// Mitsubishi GX Works2 project: PLC FX1N Program Awal Bawaan   PLC: FX1N/FX1NC

PROGRAM MAIN
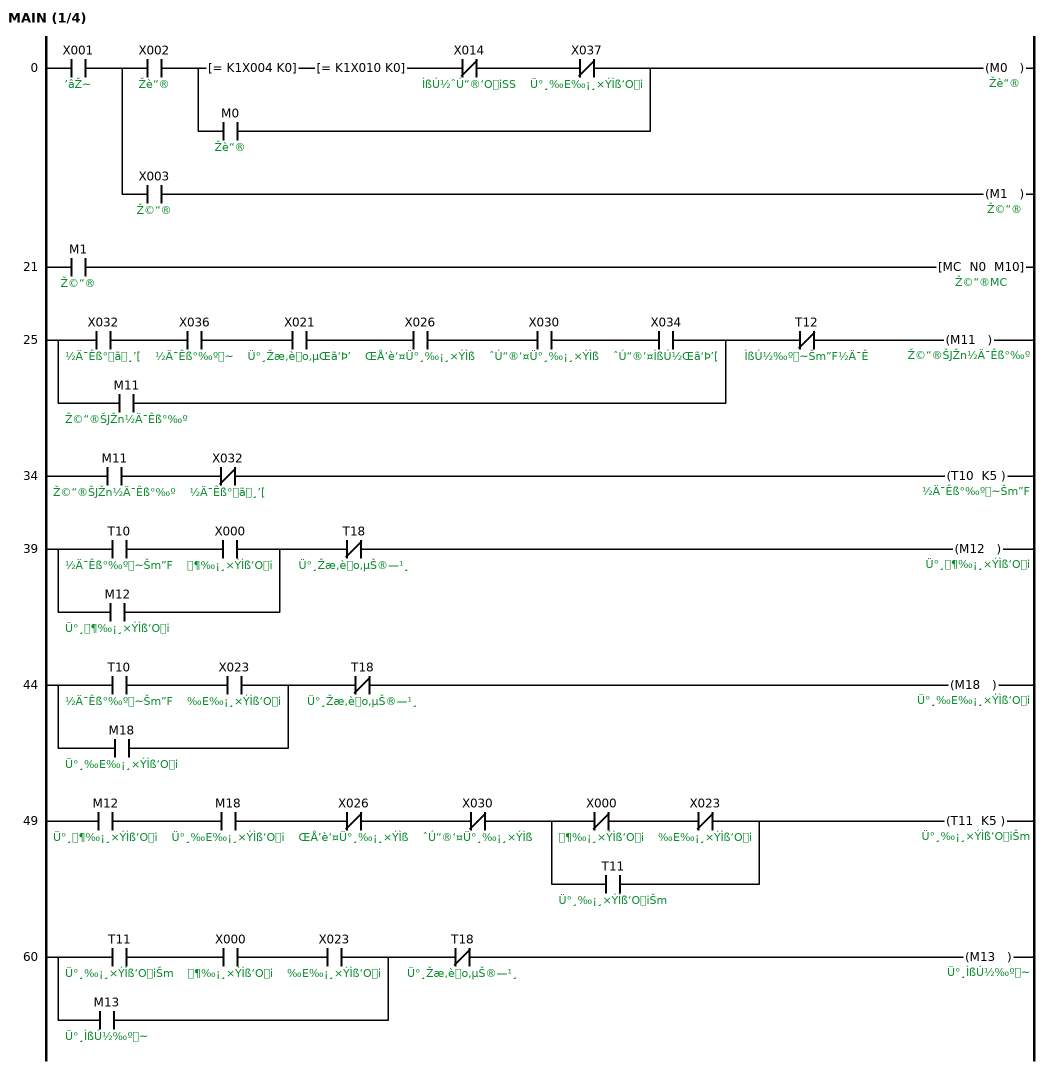
0     LD      X001  ; ’âŽ~
      MPS
      AND     X002  ; Žè“®
      LD=     K1X004 K0  ; Ü°¸Žæ‚èo‚µˆÚ“®‘
      AND=    K1X010 K0  ; ½Ä¯Êß°‰º~SS
      ANI     X014  ; ÌßÚ½ˆÚ“®‘OiSS
      ANI     X037  ; Ü°¸‰E‰¡¸×ÝÌß‘Oi
      OR      M0  ; Žè“®
      ANB
      OUT     M0  ; Žè“®
      MPP
      AND     X003  ; Ž©“®
      OUT     M1  ; Ž©“®
21    LD      M1  ; Ž©“®
      MC      N0 M10  ; Ž©“®MC
25    LD      X032  ; ½Ä¯Êß°ã¸’[
      AND     X036  ; ½Ä¯Êß°‰º~
      AND     X021  ; Ü°¸Žæ‚èo‚µŒã‘Þ’
      AND     X026  ; ŒÅ’è‘¤Ü°¸‰¡¸×ÝÌß
      AND     X030  ; ˆÚ“®‘¤Ü°¸‰¡¸×ÝÌß
      AND     X034  ; ˆÚ“®‘¤ÌßÚ½Œã‘Þ’[
      OR      M11  ; Ž©“®ŠJŽn½Ä¯Êß°‰º
      ANI     T12  ; ÌßÚ½‰º~Šm”F½Ä¯Ê
      OUT     M11  ; Ž©“®ŠJŽn½Ä¯Êß°‰º
34    LD      M11  ; Ž©“®ŠJŽn½Ä¯Êß°‰º
      ANI     X032  ; ½Ä¯Êß°ã¸’[
      OUT     T10 K5  ; ½Ä¯Êß°‰º~Šm”F
39    LD      T10  ; ½Ä¯Êß°‰º~Šm”F
      AND     X000  ; ¶‰¡¸×ÝÌß‘Oi
      OR      M12  ; Ü°¸¶‰¡¸×ÝÌß‘Oi
      ANI     T18  ; Ü°¸Žæ‚èo‚µŠ®—¹¸
      OUT     M12  ; Ü°¸¶‰¡¸×ÝÌß‘Oi
44    LD      T10  ; ½Ä¯Êß°‰º~Šm”F
      AND     X023  ; ‰E‰¡¸×ÝÌß‘Oi
      OR      M18  ; Ü°¸‰E‰¡¸×ÝÌß‘Oi
      ANI     T18  ; Ü°¸Žæ‚èo‚µŠ®—¹¸
      OUT     M18  ; Ü°¸‰E‰¡¸×ÝÌß‘Oi
49    LD      M12  ; Ü°¸¶‰¡¸×ÝÌß‘Oi
      AND     M18  ; Ü°¸‰E‰¡¸×ÝÌß‘Oi
      ANI     X026  ; ŒÅ’è‘¤Ü°¸‰¡¸×ÝÌß
      ANI     X030  ; ˆÚ“®‘¤Ü°¸‰¡¸×ÝÌß
      LDI     X000  ; ¶‰¡¸×ÝÌß‘Oi
      ANI     X023  ; ‰E‰¡¸×ÝÌß‘Oi
      OR      T11  ; Ü°¸‰¡¸×ÝÌß‘OiŠm
      ANB
      OUT     T11 K5  ; Ü°¸‰¡¸×ÝÌß‘OiŠm
60    LD      T11  ; Ü°¸‰¡¸×ÝÌß‘OiŠm
      AND     X000  ; ¶‰¡¸×ÝÌß‘Oi
      AND     X023  ; ‰E‰¡¸×ÝÌß‘Oi
      OR      M13  ; Ü°¸ÌßÚ½‰º~
      ANI     T18  ; Ü°¸Žæ‚èo‚µŠ®—¹¸
      OUT     M13  ; Ü°¸ÌßÚ½‰º~
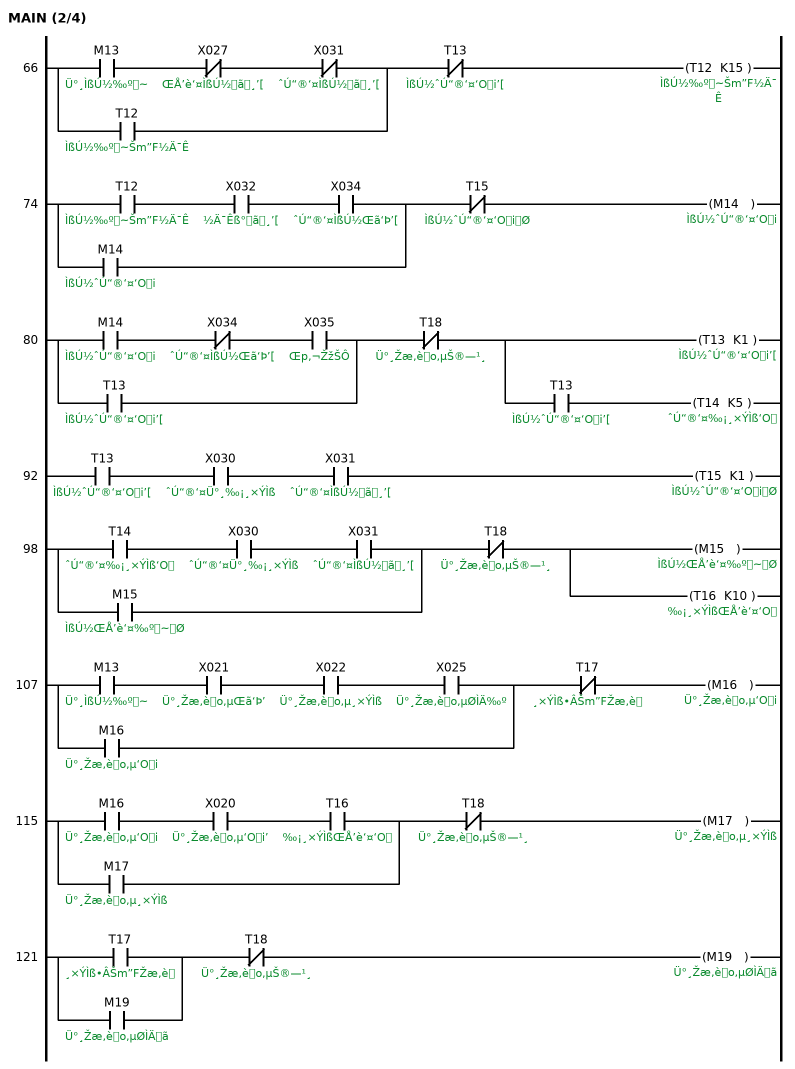
66    LD      M13  ; Ü°¸ÌßÚ½‰º~
      ANI     X027  ; ŒÅ’è‘¤ÌßÚ½ã¸’[
      ANI     X031  ; ˆÚ“®‘¤ÌßÚ½ã¸’[
      OR      T12  ; ÌßÚ½‰º~Šm”F½Ä¯Ê
      ANI     T13  ; ÌßÚ½ˆÚ“®‘¤‘Oi’[
      OUT     T12 K15  ; ÌßÚ½‰º~Šm”F½Ä¯Ê
74    LD      T12  ; ÌßÚ½‰º~Šm”F½Ä¯Ê
      AND     X032  ; ½Ä¯Êß°ã¸’[
      AND     X034  ; ˆÚ“®‘¤ÌßÚ½Œã‘Þ’[
      OR      M14  ; ÌßÚ½ˆÚ“®‘¤‘Oi
      ANI     T15  ; ÌßÚ½ˆÚ“®‘¤‘OiØ
      OUT     M14  ; ÌßÚ½ˆÚ“®‘¤‘Oi
80    LD      M14  ; ÌßÚ½ˆÚ“®‘¤‘Oi
      ANI     X034  ; ˆÚ“®‘¤ÌßÚ½Œã‘Þ’[
      AND     X035  ; Œp‚¬ŽžŠÔ
      OR      T13  ; ÌßÚ½ˆÚ“®‘¤‘Oi’[
      ANI     T18  ; Ü°¸Žæ‚èo‚µŠ®—¹¸
      OUT     T13 K1  ; ÌßÚ½ˆÚ“®‘¤‘Oi’[
      AND     T13  ; ÌßÚ½ˆÚ“®‘¤‘Oi’[
      OUT     T14 K5  ; ˆÚ“®‘¤‰¡¸×ÝÌß‘O
92    LD      T13  ; ÌßÚ½ˆÚ“®‘¤‘Oi’[
      AND     X030  ; ˆÚ“®‘¤Ü°¸‰¡¸×ÝÌß
      AND     X031  ; ˆÚ“®‘¤ÌßÚ½ã¸’[
      OUT     T15 K1  ; ÌßÚ½ˆÚ“®‘¤‘OiØ
98    LD      T14  ; ˆÚ“®‘¤‰¡¸×ÝÌß‘O
      AND     X030  ; ˆÚ“®‘¤Ü°¸‰¡¸×ÝÌß
      AND     X031  ; ˆÚ“®‘¤ÌßÚ½ã¸’[
      OR      M15  ; ÌßÚ½ŒÅ’è‘¤‰º~Ø
      ANI     T18  ; Ü°¸Žæ‚èo‚µŠ®—¹¸
      OUT     M15  ; ÌßÚ½ŒÅ’è‘¤‰º~Ø
      OUT     T16 K10  ; ‰¡¸×ÝÌßŒÅ’è‘¤‘O
107   LD      M13  ; Ü°¸ÌßÚ½‰º~
      AND     X021  ; Ü°¸Žæ‚èo‚µŒã‘Þ’
      AND     X022  ; Ü°¸Žæ‚èo‚µ¸×ÝÌß
      AND     X025  ; Ü°¸Žæ‚èo‚µØÌÄ‰º
      OR      M16  ; Ü°¸Žæ‚èo‚µ‘Oi
      ANI     T17  ; ¸×ÝÌß•ÂŠm”FŽæ‚è
      OUT     M16  ; Ü°¸Žæ‚èo‚µ‘Oi
115   LD      M16  ; Ü°¸Žæ‚èo‚µ‘Oi
      AND     X020  ; Ü°¸Žæ‚èo‚µ‘Oi’
      AND     T16  ; ‰¡¸×ÝÌßŒÅ’è‘¤‘O
      OR      M17  ; Ü°¸Žæ‚èo‚µ¸×ÝÌß
      ANI     T18  ; Ü°¸Žæ‚èo‚µŠ®—¹¸
      OUT     M17  ; Ü°¸Žæ‚èo‚µ¸×ÝÌß
121   LD      T17  ; ¸×ÝÌß•ÂŠm”FŽæ‚è
      OR      M19  ; Ü°¸Žæ‚èo‚µØÌÄã
      ANI     T18  ; Ü°¸Žæ‚èo‚µŠ®—¹¸
      OUT     M19  ; Ü°¸Žæ‚èo‚µØÌÄã
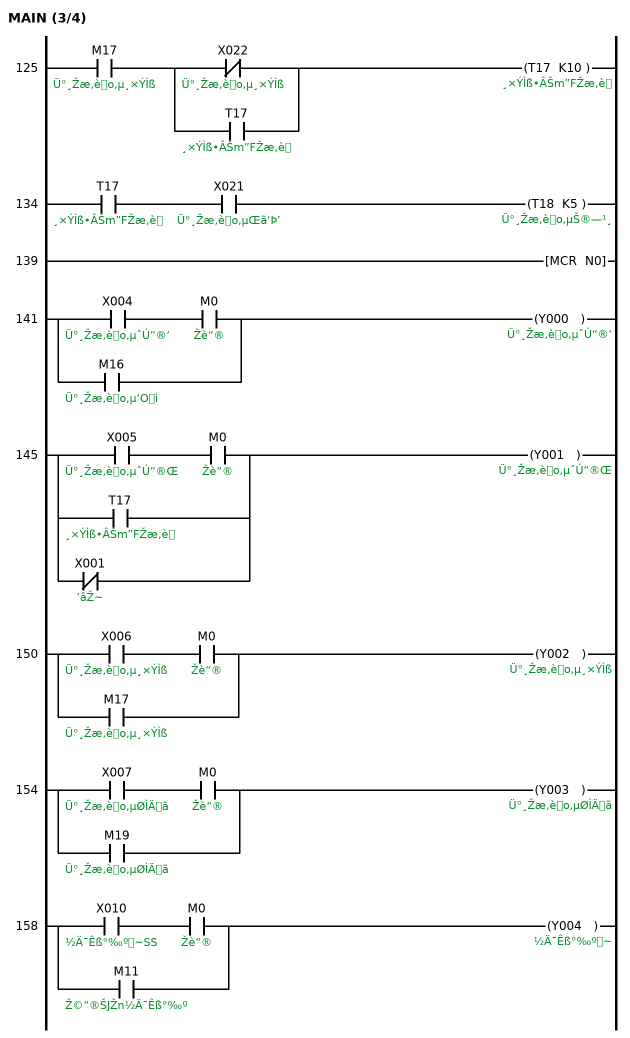
125   LD      M17  ; Ü°¸Žæ‚èo‚µ¸×ÝÌß
      LDI     X022  ; Ü°¸Žæ‚èo‚µ¸×ÝÌß
      OR      T17  ; ¸×ÝÌß•ÂŠm”FŽæ‚è
      ANB
      OUT     T17 K10  ; ¸×ÝÌß•ÂŠm”FŽæ‚è
134   LD      T17  ; ¸×ÝÌß•ÂŠm”FŽæ‚è
      AND     X021  ; Ü°¸Žæ‚èo‚µŒã‘Þ’
      OUT     T18 K5  ; Ü°¸Žæ‚èo‚µŠ®—¹¸
139   MCR     N0
141   LD      X004  ; Ü°¸Žæ‚èo‚µˆÚ“®‘
      AND     M0  ; Žè“®
      OR      M16  ; Ü°¸Žæ‚èo‚µ‘Oi
      OUT     Y000  ; Ü°¸Žæ‚èo‚µˆÚ“®‘
145   LD      X005  ; Ü°¸Žæ‚èo‚µˆÚ“®Œ
      AND     M0  ; Žè“®
      OR      T17  ; ¸×ÝÌß•ÂŠm”FŽæ‚è
      ORI     X001  ; ’âŽ~
      OUT     Y001  ; Ü°¸Žæ‚èo‚µˆÚ“®Œ
150   LD      X006  ; Ü°¸Žæ‚èo‚µ¸×ÝÌß
      AND     M0  ; Žè“®
      OR      M17  ; Ü°¸Žæ‚èo‚µ¸×ÝÌß
      OUT     Y002  ; Ü°¸Žæ‚èo‚µ¸×ÝÌß
154   LD      X007  ; Ü°¸Žæ‚èo‚µØÌÄã
      AND     M0  ; Žè“®
      OR      M19  ; Ü°¸Žæ‚èo‚µØÌÄã
      OUT     Y003  ; Ü°¸Žæ‚èo‚µØÌÄã
158   LD      X010  ; ½Ä¯Êß°‰º~SS
      AND     M0  ; Žè“®
      OR      M11  ; Ž©“®ŠJŽn½Ä¯Êß°‰º
      OUT     Y004  ; ½Ä¯Êß°‰º~
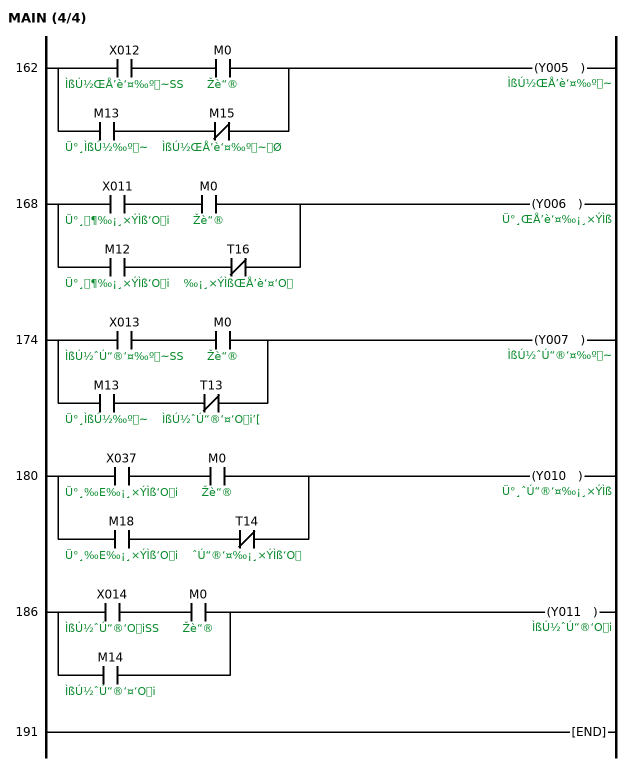
162   LD      X012  ; ÌßÚ½ŒÅ’è‘¤‰º~SS
      AND     M0  ; Žè“®
      LD      M13  ; Ü°¸ÌßÚ½‰º~
      ANI     M15  ; ÌßÚ½ŒÅ’è‘¤‰º~Ø
      ORB
      OUT     Y005  ; ÌßÚ½ŒÅ’è‘¤‰º~
168   LD      X011  ; Ü°¸¶‰¡¸×ÝÌß‘Oi
      AND     M0  ; Žè“®
      LD      M12  ; Ü°¸¶‰¡¸×ÝÌß‘Oi
      ANI     T16  ; ‰¡¸×ÝÌßŒÅ’è‘¤‘O
      ORB
      OUT     Y006  ; Ü°¸ŒÅ’è‘¤‰¡¸×ÝÌß
174   LD      X013  ; ÌßÚ½ˆÚ“®‘¤‰º~SS
      AND     M0  ; Žè“®
      LD      M13  ; Ü°¸ÌßÚ½‰º~
      ANI     T13  ; ÌßÚ½ˆÚ“®‘¤‘Oi’[
      ORB
      OUT     Y007  ; ÌßÚ½ˆÚ“®‘¤‰º~
180   LD      X037  ; Ü°¸‰E‰¡¸×ÝÌß‘Oi
      AND     M0  ; Žè“®
      LD      M18  ; Ü°¸‰E‰¡¸×ÝÌß‘Oi
      ANI     T14  ; ˆÚ“®‘¤‰¡¸×ÝÌß‘O
      ORB
      OUT     Y010  ; Ü°¸ˆÚ“®‘¤‰¡¸×ÝÌß
186   LD      X014  ; ÌßÚ½ˆÚ“®‘OiSS
      AND     M0  ; Žè“®
      OR      M14  ; ÌßÚ½ˆÚ“®‘¤‘Oi
      OUT     Y011  ; ÌßÚ½ˆÚ“®‘Oi
191   END
END_PROGRAM

// device comments not shown above
X024  ; Ü°¸Žæ‚èo‚µØÌÄã
X033  ; ˆÚ“®‘¤ÌßÚ½‘Oi’[
